{attribute 'qualified_only'}
{attribute 'strict'}
{attribute 'to_string'}
TYPE E_State :
(
	Idel:=0		,
	LoadTunningParmaeters:=1,
	AutoTuneInProgress:=2,
	LoadRunParameters:=3,
	Run:=4,
	Error:=5,
	Reset:=6
);
END_TYPE

(* stored: Version 1.1.0.1, ProductVersion 3.1.4024.12
   DUT E_State: Id {8dad1f35-ee6f-4c7c-aeed-a7b4eff901d8} *)
